FUNCTION_BLOCK Q_LockUnlockMask (* Command Lock/UnlockMask( Part 6 - F.46 ) *)
  (* Standard: ISO 11783-6; Description: Copyright (c) 2022 HR Agrartechnik GmbH This program and the accompanying materials are made available under the terms of the Eclipse Public License 2.0 which is available at https://www.eclipse.org/legal/epl-2.0/ SPDX-License-Identifier: EPL-2.0 see Description Tab *)
  (* Version 1.0, 2022-07-08, Franz Höpfinger, HR Agrartechnik GmbH *)
  PACKAGE isobus::UT::Q;
  IMPORT eclipse4diac::core::TypeHash;
  IMPORT isobus::UT::Q::IDs::ID_NULL;
  (* Documentation:
  Command Lock/UnlockMask( Part 6 - F.46 )
   This message is available in VT Version 4 and later. This command is used by a Working Set to disallow or allow screen refreshes at the VT for the visible Data Mask or User-Layout Data Mask owned by the requesting Working Set.
   param[in] {state, uint8_t}
   0 = Unlock, 1 = Lock data mask or user-layout data mask
   param[in] {objectID,  uint16_t}
   Object ID of data mask or user layout data mask to lock or unlock
   param[in] {timeout_ms,  uint16_t}
   Lock timeout in ms or zero for no timeout
   Return Values: 
   int16_t
    - VT_E_NO_ERR (0) - OK
   - VT_E_OVERFLOW (-6) - buffer overflow
   - VT_E_NOACT (-8) - Command not possible in current state
   - VT_E_NO_INSTANCE (-21) - No VT client available
   - VT_E_ISO_INSTANCE_INVALID (-129) - Identifier for instance (connection) invalid
   - VT_E_NOT_ALIVE (-130) - Identifier for instance valid, but VT Dead.
  *)
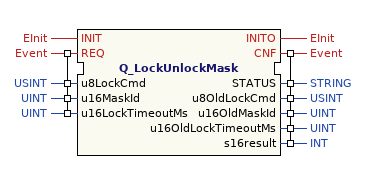
  EVENT_INPUT
    INIT : EInit; (* Service Initialization *)
    REQ WITH u8LockCmd, u16MaskId, u16LockTimeoutMs; (* Service Request *)
  END_EVENT
  EVENT_OUTPUT
    INITO : EInit; (* Initialization Confirm *)
    CNF WITH STATUS, s16result, u8OldLockCmd, u16OldMaskId, u16OldLockTimeoutMs; (* Confirmation of Requested Service *)
  END_EVENT
  VAR_INPUT
    u8LockCmd : USINT; (* 0 = Unlock, 1 = Lock data mask or user-layout data mask *)
    u16MaskId : UINT := ID_NULL; (* Object ID of data mask or user layout data mask to lock or unlock *)
    u16LockTimeoutMs : UINT; (* Lock timeout in ms or zero for no timeout *)
  END_VAR
  VAR_OUTPUT
    STATUS : STRING; (* Service Status *)
    u8OldLockCmd : USINT; (* Old 0 = Unlock, 1 = Lock data mask or user-layout data mask *)
    u16OldMaskId : UINT; (* Old object ID of data mask or user layout data mask to lock or unlock *)
    u16OldLockTimeoutMs : UINT; (* Old lock timeout in ms or zero for no timeout *)
    s16result : INT; (* retval see description *)
  END_VAR
END_FUNCTION_BLOCK
